// Fail is the outright failure with no comparison behind it - for a branch that
// should have been unreachable. It is a Failed verdict, not an Errored one:
// reaching that branch IS the code being wrong.
FUNCTION_BLOCK TEST_VerdictFailIsAPlainFailure IMPLEMENTS I_Test
VAR
	// A private journal and handle, so a DELIBERATE failure can be recorded and
	// inspected without the suite's own verdict ever seeing it. The test itself
	// passes; what it proves is that failing works.
	Subject : TestJournal;
	Handle	: TestVerdict;
	ExpectedStatus : E_TestStatus;
	ActualStatus   : E_TestStatus;
END_VAR

METHOD Run : BOOL
VAR_INPUT
	Enable : BOOL;
	Test   : I_TestAssertions;
END_VAR
Handle.Target(Subject);
Subject.Begin('unreachable branch', '');

Handle.Fail('the default case was reached');

Subject.Finish(E_TestStatus.Passed);

ExpectedStatus := E_TestStatus.Failed;
ActualStatus   := Subject.Status;
Test.AssertEqual(ExpectedStatus, ActualStatus, 'Fail produces Failed');

Handle.Untarget();

Run := TRUE;
END_METHOD

END_FUNCTION_BLOCK

(* stored: Version 1.1.0.1, ProductVersion 3.1.4026.18
   POU TEST_VerdictFailIsAPlainFailure: Id {9b398a39-71b5-4057-9a95-df7334a37f86}, SpecialFunc None
   Folder I_Test: Id {2071e105-cfaa-4b19-9395-0c503871afd5}
   Method Run: Id {fe0f0e62-4159-4537-9aec-73bd64dd2ec8} *)
